// TIA Portal V18 export
DATA_BLOCK "artLimFormer_DB"   // DB73
VERSION : 0.1
// stored: AutoNumber true, DBAccessibleFromOPCUA true, InstanceOfName artLimFormer, InstanceOfType FB
"artLimFormer"
   // VAR_INPUT
   //    doors_open_fully : Bool := FALSE;
   //    pos_x : Real := 0.0;
   //    pos_y : Real := 0.0;
   //    lim_yrev_chamber_doorsClosed_safe : Real := -20.0;
   //    lim_x_fwd_outside : Real := 50.0;
   //    lim_x_rev_outside : Real := -50.0;
   //    normal_x_rev : Real := -200.0;
   //    normal_x_fwd : Real := 200.0;
   //    normal_y_rev : Real := -4400.0;
   //    normal_y_fwd : Real := 4440.0;
   //    margin_x : Real := 5.0;
   //    ACK : Bool := FALSE;
   //    margin_y : Real := 5.0;
   // END_VAR
   // VAR_OUTPUT
   //    result_x_rev : Real;
   //    result_x_fwd : Real;
   //    result_y_rev : Real;
   //    result_y_fwd : Real;
   //    ER_WS : WString := WSTRING#'';
   //    ER : Bool := FALSE;
   //    y_is_inside_safely : Bool := FALSE;
   // END_VAR
   // VAR
   //    y_can_go_out_rev : Bool := FALSE;
   //    x_fits_in_doors : Bool := TRUE;
   //    y_is_inside : Bool := TRUE;
   // END_VAR
BEGIN
END_DATA_BLOCK
